// TIA Portal V19 export
DATA_BLOCK "P TRIG"   // DB115
{ S7_Optimized_Access := 'TRUE' }
// stored: MemoryReserve 100
   VAR
      P_TRIG : Struct
         "1" : Bool;
         "2" : Bool;
         "3" : Bool;
         "4" : Bool;
         "5" : Bool;
         "6" : Bool;
         "7" : Bool;
         "8" : Bool;
         "9" : Bool;
         "10" : Bool;
         "11" : Bool;
         "12" : Bool;
         "13" : Bool;
         "14" : Bool;
         "15" : Bool;
         "16" : Bool;
         "17" : Bool;
         "18" : Bool;
         "19" : Bool;
         "20" : Bool;
         "21" : Bool;
         "22" : Bool;
         "23" : Bool;
         "24" : Bool;
         "25" : Bool;
         "26" : Bool;
         "27" : Bool;
         "28" : Bool;
         "29" : Bool;
         "30" : Bool;
         "31" : Bool;
         "32" : Bool;
         "33" : Bool;
         "34" : Bool;
         "35" : Bool;
         "36" : Bool;
         "37" : Bool;
         "38" : Bool;
         "39" : Bool;
         "40" : Bool;
         "41" : Bool;
         "42" : Bool;
         "43" : Bool;
         "44" : Bool;
         "45" : Bool;
         "46" : Bool;
         "47" : Bool;
         "48" : Bool;
         "49" : Bool;
         "50" : Bool;
         "51" : Bool;
         "52" : Bool;
         "53" : Bool;
         "54" : Bool;
         "55" : Bool;
         "56" : Bool;
         "57" : Bool;
         "58" : Bool;
         "59" : Bool;
         "60" : Bool;
      END_STRUCT;
   END_VAR
BEGIN
END_DATA_BLOCK
